Staubli VAL3: Palacinke.pjx

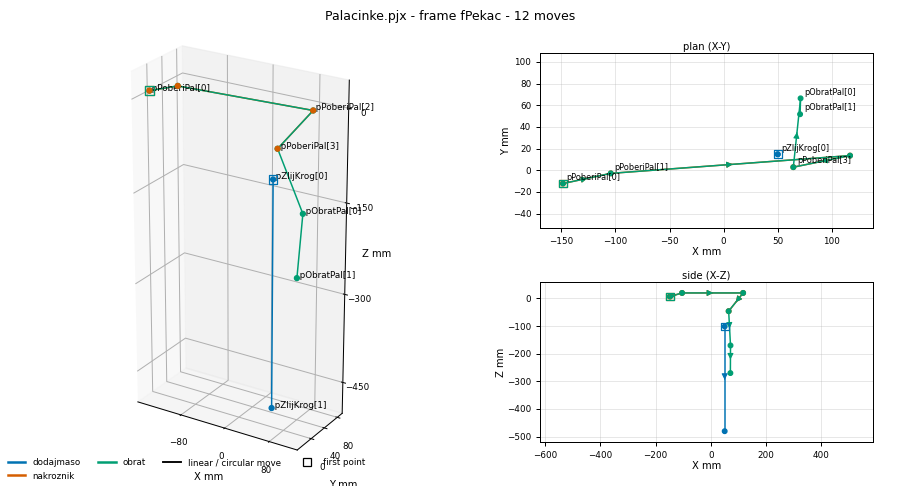
[picture p0: tool path of Palacinke.pjx in frame fPekac, 12 of 32 moves have a stored position in this frame; points joined in program order, loops and branches not executed]
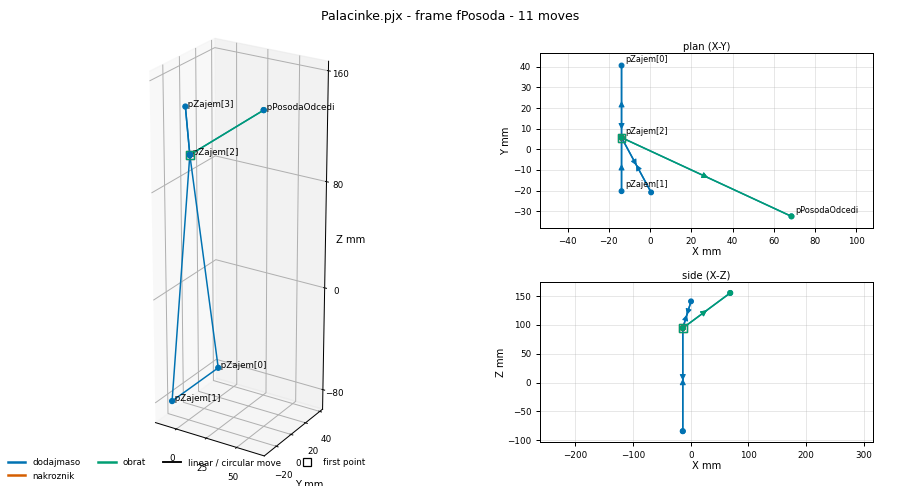
[picture p1: tool path of Palacinke.pjx in frame fPosoda, 11 of 32 moves have a stored position in this frame; points joined in program order, loops and branches not executed]
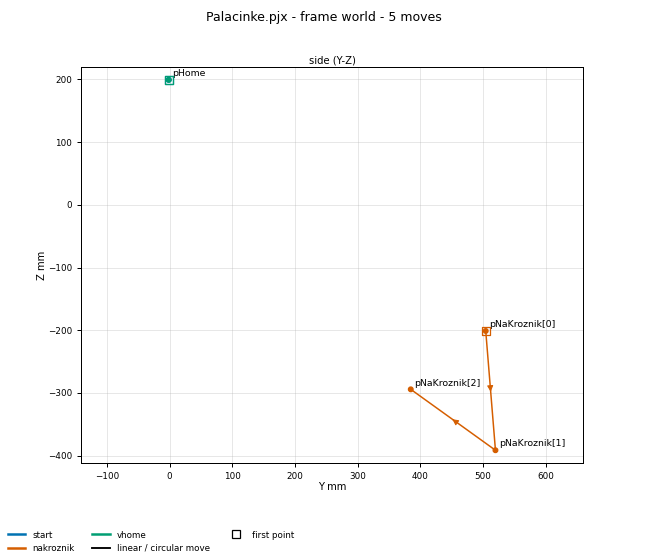
[picture p2: tool path of Palacinke.pjx in frame world, 5 of 32 moves have a stored position in this frame; points joined in program order, loops and branches not executed]
--- Palacinke.pjx ---
Parameters version=s8.15.3Cs9_BS3337 stackSize=20000 millimeterUnit=true
Program file=avtomatskiCikel.pgx
Program file=cakajProgress.pgx
Program file=DodajMaso.pgx
Program file=Glavni.pgx
Program file=naKroznik.pgx
Program file=obrat.pgx
Program file=reset.pgx
Program file=safety.pgx
Program file=start.pgx
Program file=stop.pgx
Program file=taski.pgx
Program file=vHome.pgx
Data file=Palacinke.dtx

--- Palacinke.dtx ---
configRx cConfigHome = {shoulder=lefty, elbow=epositive, wrist=wfree}
frame fPekac = {x=490, y=110.0000152588, z=-315, rx=-179.999991, ry=-8.53774E-06, rz=-46.970374, fatherId=world[0]}
frame fPosoda = {x=276.386063, y=-415.101207, z=-289.00196368, rx=9.03224E-05, ry=-0.0274943, rz=-0.013391, fatherId=world[0]}
frame fSist = {x=112.012468, y=457.500263, z=-311.848898, rz=-15, fatherId=world[0]}
jointRx jHome = {j1=-3.713051, j2=4.261033, j3=89.403973, j4=4.2726E-05, j5=86.333741, j6=139.618635}
jointRx jNadPosodo = {j1=-47.707914, j2=16.909947, j3=91.537983, j4=27.468698, j5=86.330149, j6=139.620943}
jointRx jTrenutna = {j1=-3.714387, j2=4.262257, j3=89.411972, j4=-0.00277969, j5=86.334942, j6=139.61472}
mdesc mHitro = {accel=70, vel=70, decel=50, leave=80, reach=80}
mdesc mNomSpeed = {tmax=10, rmax=10}
mdesc mPocasi = {accel=50, vel=70, decel=50, tmax=80, rmax=80, leave=5, reach=5}
mdesc mSrednje = {accel=90, decel=90, tmax=110, rmax=110, leave=30, reach=30}
num nCas_peke1 = 95
num nCas_peke2 = 76
num nCounter
num nGumb = 1
pointRx pHome = {x=331.509669, y=-1.48229, z=199.354371, rx=-179.999362, ry=-0.00397297, rz=-36.668093, shoulder=lefty, elbow=epositive, wrist=wfree, fatherId=world[0]}
pointRx pNaKroznik[3]
  [0] = {x=327.514302, y=504.0779887, z=-201.12708, rx=-5.275089, ry=-0.617248, rz=91.137777, shoulder=lefty, elbow=epositive, wrist=wpositive, fatherId=world[0]}
  [1] = {x=327.51452, y=519.577474, z=-391.392589, rx=-33.60943, ry=-0.616673, rz=91.138436, shoulder=lefty, elbow=epositive, wrist=wpositive, fatherId=world[0]}
  [2] = {x=327.514234, y=384.497454, z=-294.236732, rx=-58.82704, ry=-0.616669, rz=91.13839, shoulder=lefty, elbow=epositive, wrist=wpositive, fatherId=world[0]}
pointRx pNadPekac = {x=-73.960476, y=-46.850855, z=-190.433189, rx=24.649117, ry=43.0990687, rz=131.714196, shoulder=sfree, elbow=efree, wrist=wfree, fatherId=fPekac[0]}
pointRx pObratPal[2]
  [0] = {x=71.0587127, y=66.364886, z=-170.0723603, rx=-179.779763, ry=5.303293, rz=-7.926087, shoulder=lefty, elbow=epositive, wrist=wpositive, fatherId=fPekac[0]}
  [1] = {x=70.605667, y=51.703876, z=-270.0649837, rx=71.732423, ry=6.792126, rz=6.715035, shoulder=lefty, elbow=epositive, wrist=wpositive, fatherId=fPekac[0]}
pointRx pPoberiPal[4]
  [0] = {x=-148.41772, y=-12.314447, z=6.994822, rx=170.48509, ry=32.610293, rz=-4.244789, shoulder=lefty, elbow=epositive, wrist=wpositive, fatherId=fPekac[0]}
  [1] = {x=-104.25102, y=-2.921622, z=19.963319, rx=170.484931, ry=32.60972, rz=-4.245238, shoulder=lefty, elbow=epositive, wrist=wpositive, fatherId=fPekac[0]}
  [2] = {x=116.744491, y=13.47581, z=19.984953, rx=177.965469, ry=12.205717, rz=-7.661892, shoulder=lefty, elbow=epositive, wrist=wpositive, fatherId=fPekac[0]}
  [3] = {x=64.359214, y=2.794031, z=-46.0313774, rx=178.00569366, ry=4.309998, rz=-7.942312, shoulder=lefty, elbow=epositive, wrist=wpositive, fatherId=fPekac[0]}
pointRx pPosodaOdcedi = {x=68.501243, y=-32.472804, z=155.463999, rx=-44.507181, ry=45.37821, rz=-5.856988, shoulder=lefty, elbow=epositive, wrist=wpositive, fatherId=fPosoda[0]}
pointRx pZajem[4]
  [0] = {x=-13.832248, y=40.613124, z=-84.448672, rx=59.615179, ry=165.914626, rz=-87.31672, shoulder=lefty, elbow=epositive, wrist=wpositive, fatherId=fPosoda[0]}
  [1] = {x=-13.832408, y=-20.27955, z=-84.448613, rx=59.614116, ry=165.914404, rz=-87.316919, shoulder=lefty, elbow=epositive, wrist=wpositive, fatherId=fPosoda[0]}
  [2] = {x=-13.832691, y=5.683948, z=94.444293, rx=39.32001, ry=171.222369, rz=-87.991671, shoulder=lefty, elbow=epositive, wrist=wpositive, fatherId=fPosoda[0]}
  [3] = {x=0.494953, y=-20.859447, z=140.876688, rx=54.411966, ry=171.221555, rz=-87.992016, shoulder=lefty, elbow=epositive, wrist=wpositive, fatherId=fPosoda[0]}
pointRx pZlijKrog[4]
  [0] = {x=49.976213, y=14.693648, z=-101.351585, rx=31.529296, ry=15.883124, rz=100.846893, shoulder=lefty, elbow=epositive, wrist=wpositive, fatherId=fPekac[0]}
  [1] = {x=49.976117, y=14.693627, z=-480.425915, rx=139.262761, ry=38.958791, rz=-44.051028, shoulder=lefty, elbow=epositive, wrist=wpositive, fatherId=fPekac[0]}
  [2] = {x=38.327918, y=75.963557, z=-105.369298, rx=-100.0134396, ry=-16.583777, rz=-25.943731, shoulder=lefty, elbow=epositive, wrist=wpositive, fatherId=fPekac[0]}
  [3] = {x=33.00287087, y=-6.527576, z=-94.55238, rx=-100.284225, ry=-16.610358, rz=-26.0271264, shoulder=lefty, elbow=epositive, wrist=wpositive, fatherId=fPekac[0]}
string sDiag = "Robot ustavljen zaradi odprtih vrat"
tool tLopatka = {x=240, z=90, rx=-180, fatherId=flange[0], ioLink=ValveIO\valve1}
tool tOrodje = {y=230, z=100, rz=90, fatherId=flange[0], ioLink=ValveIO\valve1}
tool tSefla = {y=230, z=100, rz=90, fatherId=flange[0], ioLink=ValveIO\valve1}
num nProgress
num nTaskWorking = 1

--- start.pgx ---
program start()
begin

  userPage("pala_cinke")
  call cakajProgress(1)
  enablePower()
  setMonitorSpeed(50)

  taskCreate "Safety",80,safety()

  movej(pHome,flange,mSrednje)

  // Ali robot izvaja (pekalni) task
  nTaskWorking = 0
  // Čas peke (Čas1 = čas pečenja na prvi strani)
  nCas_peke1=95
  nCas_peke2=nCas_peke1*0.8

  do
    jTrenutna=herej()
  until false
end

--- avtomatskiCikel.pgx ---
program avtomatskiCikel()
begin

  // neskončna zanka pečenja palačink

  do
  //  call DodajMaso()
    //sDiag="Pečem prvo stran"
   // delay(nCas_peke1)
    //call obrat()
    //sDiag="Pečem drugo stran"
    //delay(nCas_peke2)
    //call naKroznik()
    call Glavni()
  until false
end

--- cakajProgress.pgx ---
program cakajProgress(num x_nCas)
  local num l_nNuml_nStartTime
  local num l_nTimeRazlika
  local num l_nStartTime
begin
  // cakajProgress
  // @param x_nCas(num)  Funkcija resetira progress bar in s pomocjo razlike
  // casa prek clock() funkcije steje koliko casa je preostalo do konca, medtem ko
  // posodablja progress bar (nProgress) na grafičnem vmesniku

  // Resetiraj progress display
  nProgress = 0
  // Postavi casovno razliko na 0
  l_nTimeRazlika = 0
  // Trenutno pretekle sekunde
  l_nStartTime = clock()
  while l_nTimeRazlika < x_nCas
    delay(0.1)
    l_nTimeRazlika = clock() - l_nStartTime
    nProgress = min(100*l_nTimeRazlika/x_nCas, 100)
  endWhile
end

--- DodajMaso.pgx ---
program DodajMaso()
  local num l_ni
begin

  // TUKAJ vstavi ukaze za premikanje robota na krožnik
  // lahko si pomagaš s starimi točkami, ki so tu spodaj zakomentirane

  // namesto mNomSpeed uporabi že pripravljene hitrosti mPočasi, mSrednje in mHitro, glede na to kakšno gibanje želiš
  // ukaz waitEndMove uporabimo, ko želimo, da se robot v vsaki točki ustavi. Ko se pomikamo po prostoru, ne želimo ustavljanja preko vseh točk, ampak želimo zvezno gibanje
  // v definiciji vsake hitrosti je tudi možnost blend, ki pove koliko milimetrov od točke naj potuje robot, ko gre proti naslednji brez ustavljanja
  // če želimo točne pomike, za primer pobiranja, uporabimo waitEndMove, da se robot pomakne točno v točko in tam počaka na naslednji ukaz

  // če podatek ni shranjen kot array (ima le indeks [0]), ga lahko kličemo le z imenom, brez indeksa. Če imamo array z več vnosi/indeksi pa na ta način kličemo ničti [0] element.
  // primer: mNomSpeed[0] == mNomSpeed

  nTaskWorking = nTaskWorking + 1
  movel(pZajem[2],tSefla,mSrednje)
  movel(pZajem[0],tSefla,mPocasi)
  movel(pZajem[1],tSefla,mPocasi)
  movel(pZajem[2],tSefla,mPocasi)
  waitEndMove()

  for l_ni=0 to 4
    movel(pZajem[3],tSefla,mHitro)
    waitEndMove()
    movel(pZajem[2],tSefla,mHitro)
    waitEndMove()
  endFor

  call cakajProgress(8)


  movel(pZlijKrog[0],tSefla,mSrednje)
  movel(pZlijKrog[1],tSefla,mPocasi)
  waitEndMove()
  call cakajProgress(10)

  movel(pZajem[2],tSefla,mSrednje)
  movel(pPosodaOdcedi,tSefla,mSrednje)
  waitEndMove()
  nTaskWorking = nTaskWorking - 1
end

--- Glavni.pgx ---
program Glavni()
begin

  // pečenje samo ene palačinke

  // movej(ji,tSefla,mNomSpeed) ??

  if isSettled()
    nTaskWorking[0] = nTaskWorking[0] + 1
    call cakajProgress(1)
    call DodajMaso()
    sDiag="Peka"
    // Posodabljaj progress bar in cakaj dokler je minulu manh od nCas_peke1
    call cakajProgress(nCas_peke1)
    call obrat()
    sDiag="Peka"
    // Posodabljaj progress bar in cakaj dokler je minulu manh od nCas_peke2
    call cakajProgress(nCas_peke2)
    call naKroznik()
    // Povecaj stevec narejenih palacinke
    nCounter = nCounter + 1
    nTaskWorking[0] = nTaskWorking[0] - 1
  endIf
end

--- naKroznik.pgx ---
program naKroznik()
begin

  // TUKAJ vstavi ukaze za premikanje robota na krožnik
  // lahko si pomagaš s starimi točkami, ki so tu spodaj zakomentirane

  // namesto mNomSpeed uporabi že pripravljene hitrosti mPočasi, mSrednje in mHitro, glede na to kakšno gibanje želiš
  // ukaz waitEndMove uporabimo, ko želimo, da se robot v vsaki točki ustavi. Ko se pomikamo po prostoru, ne želimo ustavljanja preko vseh točk, ampak želimo zvezno gibanje
  // v definiciji vsake hitrosti je tudi možnost blend, ki pove koliko milimetrov od točke naj potuje robot, ko gre proti naslednji brez ustavljanja
  // če želimo točne pomike, za primer pobiranja, uporabimo waitEndMove, da se robot pomakne točno v točko in tam počaka na naslednji ukaz

  // če podatek ni shranjen kot array (ima le indeks [0]), ga lahko kličemo le z imenom, brez indeksa. Če imamo array z več vnosi/indeksi pa na ta način kličemo ničti [0] element.
  // primer: mNomSpeed[0] == mNomSpeed

  nTaskWorking = nTaskWorking + 1

  movej(jNadPosodo,flange,mSrednje)
  waitEndMove()

  movel(pPoberiPal[0],tLopatka,mSrednje)
  movel(pPoberiPal[1],tLopatka,mSrednje)
  movel(pPoberiPal[2],tLopatka,mPocasi)
  movel(pPoberiPal[3],tLopatka,mPocasi)

  movel(pNaKroznik[0],tLopatka,mPocasi)
  movel(pNaKroznik[1],tLopatka,mPocasi)
  movel(pNaKroznik[2],tLopatka,mSrednje)
  waitEndMove()
  call cakajProgress(3)

  movej(jHome,flange,mSrednje)
  movel(pZajem[2],tSefla,mSrednje)
  waitEndMove()

 nTaskWorking = nTaskWorking - 1
end

--- obrat.pgx ---
program obrat()
begin

  // TUKAJ vstavi ukaze za premikanje robota na krožnik
  // lahko si pomagaš s starimi točkami, ki so tu spodaj zakomentirane

  // namesto mNomSpeed uporabi že pripravljene hitrosti mPočasi, mSrednje in mHitro, glede na to kakšno gibanje želiš
  // ukaz waitEndMove uporabimo, ko želimo, da se robot v vsaki točki ustavi. Ko se pomikamo po prostoru, ne želimo ustavljanja preko vseh točk, ampak želimo zvezno gibanje
  // v definiciji vsake hitrosti je tudi možnost blend, ki pove koliko milimetrov od točke naj potuje robot, ko gre proti naslednji brez ustavljanja
  // če želimo točne pomike, za primer pobiranja, uporabimo waitEndMove, da se robot pomakne točno v točko in tam počaka na naslednji ukaz

  // če podatek ni shranjen kot array (ima le indeks [0]), ga lahko kličemo le z imenom, brez indeksa. Če imamo array z več vnosi/indeksi pa na ta način kličemo ničti [0] element.
  // primer: mNomSpeed[0] == mNomSpeedW
  nTaskWorking = nTaskWorking + 1

  movej(jNadPosodo,flange,mSrednje)
  waitEndMove()

  movel(pPoberiPal[0],tLopatka,mSrednje)
  movel(pPoberiPal[1],tLopatka,mSrednje)
  movel(pPoberiPal[2],tLopatka,mSrednje)
  movel(pPoberiPal[3],tLopatka,mPocasi)
  movel(pObratPal[0],tLopatka,mPocasi)
  movel(pObratPal[1],tLopatka,mHitro)
  waitEndMove()
  call cakajProgress(3)

  movel(pZajem[2],tSefla,mSrednje)
  movel(pPosodaOdcedi,tSefla,mSrednje)
  waitEndMove()

  nTaskWorking = nTaskWorking - 1
end

--- reset.pgx ---
program reset()
  local num ln_task_i
begin

  // najprej ustavimo gibanje robota, pobrišemo vse naslednje gibe, ki bi se morali zgoditi in končamo vsa opravila
  taskKill("palacinka")
  taskKill("masa")
  taskKill("obrat")
  taskKill("kroznik")
  taskKill("samodejno")
  taskKill("home")
  stopMove()
  resetMotion()
  waitEndMove()
  call cakajProgress(1)

  // Ugasnili smo vse "glavne" taske, tako da lahko to spremenljivko nastavimo na 0,
  // s čimer spet dovolimo da se v taski() podprogramu naredi nov task
  nTaskWorking = 0
end

--- safety.pgx ---
program safety()
  local bool l_brestart
begin

  // TASK KI SKRBI ZA VARNOST - TEGA TASKA NIKOLI NE PREKINJAŠ
  // tu ne spreminjaj ničesar
  // če odpremo vrata ali pritisnemo rdeč Emergency STOP gumb, se robot ustavi
  // ko zapremo vrata se aplikacija samodejno nadaljuje kjer smo jo ustavili

  do

    // če je safety status 2, se je robot zaustavil zaradi odprtih vrat
    // ko zapremo vrata, se status nastavi na 0 in ob potrditvi nadaljujemo program

    switch esStatus()

      //vse ok
      case 0
      break

      //reset, ko sprostimo E-STOP tipko
      case 1
        sDiag="Robot ustavljen zaradi pritiska gumba"
        l_brestart=userPageConfirm("Restartam?")
        if (l_brestart)
          setSafetyRestart()
          sDiag="Varni restart JE USPEL"
          enablePower()
          stopMove()
          resetMotion()
          sDiag="Gibanje je ustavljeno in resetirano"
        else
          sDiag="Varni restart NI USPEL"
        endIf
      break

      // če se je zgodil safety stop
      case 2

        sDiag="Robot ustavljen zaradi odprtih vrat"

        //v primeru, da stisnemo E-STOP je esSafety=2 do sprostitve gumba, ko je potreben nadaljni reset
        //v nasprotnem primeru so bila odprta vrata

        wait(esStatus()==0 or esStatus()==1)
        if esStatus()==0
          sDiag="Nadaljujem!"
          enablePower()
          sDiag="Robot je varen za uporabo."
        else
          sDiag="Zapri vrata, da lahko nadaljujem!"
        endIf
      break
    endSwitch
  until false

end

--- stop.pgx ---
program stop()
begin

  stopMove()
  resetMotion()
  disablePower()
  userPage("new1")
  call cakajProgress(2)
end

--- taski.pgx ---
program taski()
begin

  // glede na to kateri gumb pritisnemo na uporabniškemu umesniku, začnemo novo opravilo
  // taske uporabljamo zato, da vsakič ko pritisnemo reset, končamo vsa opravila in se vsi ukazi gibanja pobrišejo, robot pa se ustavi in lahko gre po varni poti v home

  if isPowered()
    // Ne naredi novega taska, ce eden ze deluje
    // nTaskWorking se pristeje vsakic ko se zacne izvajati eden od "pravih" podprogramov
    // in odsteje ko se eden od podprogramov neha izvajati
    // Posledično mora biti nTaskWorking enako 0, zato da zagotovo ni v nobenem podprogramu
    if nTaskWorking > 0 and nGumb != 2
      return
    endIf

    switch nGumb
      case 1
        sDiag="Peka ene palačinke"
        taskCreate "palacinka",40,Glavni()
      break

      case 2
        sDiag="Ustavljam gibanje"
        call reset()
      break

      case 3
        sDiag="Vlivam maso na ponev"
        taskCreate "masa",40,DodajMaso()
      break

      case 4
        sDiag="Obračam"
        taskCreate "obrat",40,obrat()
      break

      case 5
        sDiag="Prenašam palačinko na krožnik"
        taskCreate "kroznik",40,naKroznik()
      break

      case 6
        sDiag="Avtomatska peka palačink"
        taskCreate "samodejno",40,avtomatskiCikel()
      break

      case 7
        sDiag="Grem v osnovni položaj"
        taskCreate "home",40,vHome()
      break

      default
      break

    endSwitch

  else
    sDiag="POZOR! Ni varno za peko palačink"
  endIf
end

--- vHome.pgx ---
program vHome()
  local pointRx l_pHome
  local pointRx l_pLokalnoGor
begin
  nTaskWorking = nTaskWorking + 1
  //l_pHome=jointToPoint(flange,world,jHome)
  cConfigHome=pHome.config
  l_pLokalnoGor=here(flange, world)
  // Vedno premakni za visino 60mm
  // Ni pomembno katero orodje je izbrano saj se premikamo po smereh globalnega sistemu
  // Orodje je pomembno tu le za dolocanje trenutne pozicija, a ni vazno kaj izberemo
  // saj orientacije ne bomo spreminjali, prav tako pa je premik relativen oz. je
  // RAZLIKA v visini ENAKA, ne glede na to katero orodje je izbrano
  l_pLokalnoGor.trsf.z= l_pLokalnoGor.trsf.z + 60
  l_pLokalnoGor={l_pLokalnoGor.trsf,cConfigHome}
  movel(l_pLokalnoGor,flange,mSrednje)
  waitEndMove()
  movel(pHome,flange,mSrednje)
  waitEndMove()
  sDiag="Sem v osnovnem položaju"
  nTaskWorking = nTaskWorking - 1
end
